{attribute 'linkalways'} 
{attribute 'no_explicit_call' := 'This FB is a CLASS and must be accessed using methods or properties'}
{attribute 'enable_dynamic_creation'}
FUNCTION_BLOCK FINAL GT_DINT EXTENDS Node
VAR
	in1 : _DINT(0);
	in2 : _DINT(0);
	out : _BOOL(FALSE);
END_VAR

METHOD PUBLIC Clone : I_Node
VAR
	pNode : POINTER TO GT_DINT;
END_VAR
pNode := __NEW(GT_DINT);
Clone := pNode^;
END_METHOD

METHOD FB_init : BOOL
VAR_INPUT
	bInitRetains : BOOL; // if TRUE, the retain variables are initialized (warm start / cold start)
	bInCopyCode : BOOL;  // if TRUE, the instance afterwards gets moved into the copy code (online change)
END_VAR
AddInput('in1',THIS^.in1);
AddInput('in2',THIS^.in2);
AddOutput('out', THIS^.out);
END_METHOD

METHOD PROTECTED OnExecute
VAR
END_VAR
out.Value := in1.Value > in2.Value;
END_METHOD

END_FUNCTION_BLOCK

(* stored: Version 1.1.0.1, ProductVersion 3.1.4024.15
   POU GT_DINT: Id {e26a6cd3-f3a0-451b-bc71-e30d601448e6}, SpecialFunc None
   Folder Constructor: Id {c250bced-a088-4523-aa78-78ab654c4c44}
   Method Clone: Id {0f3180ee-e216-47dd-ab54-ba1a5a808806}
   Method FB_init: Id {6bc1891c-ab7d-411c-9600-840707c3367d}
   Method OnExecute: Id {3e9a1e7b-5b20-42fe-9e82-1937a07851e9} *)
